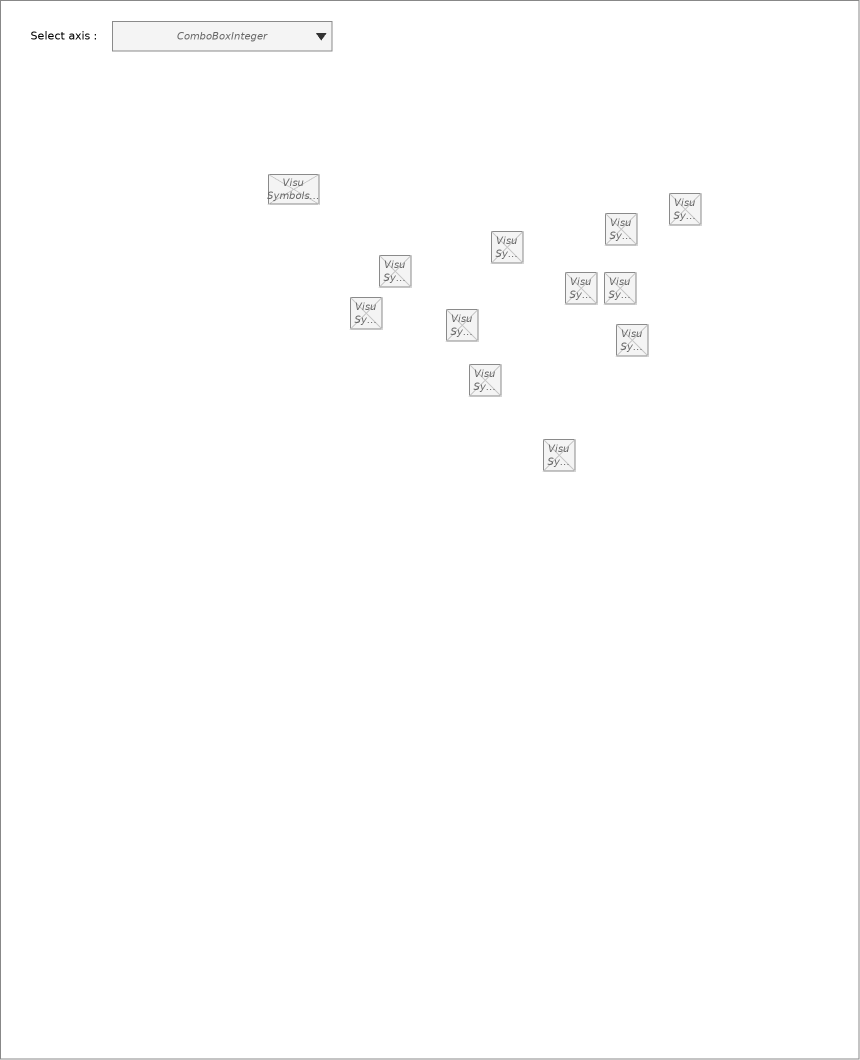
VISUALIZATION VISU_AxisManual  // 860x1060
    Label (22,21 84x30), "Select axis :"
    ComboBoxInteger (112,21 220x30), variable: HMI.iSelectJogAxis
    Image (268,174 51x30), image: VisuSymbols.Symbols.ForwardStandard
    Image (350,297 32x32), image: VisuSymbols.Symbols.Home
    Image (469,364 32x32), image: VisuSymbols.Symbols.Humidity
    Image (543,439 32x32), image: VisuSymbols.Symbols.Keeper
    Image (446,309 32x32), image: VisuSymbols.Symbols.ListNumbers
    Image (604,272 32x32), image: VisuSymbols.Symbols.Marker+
    Image (565,272 32x32), image: VisuSymbols.Symbols.Marker-
    Image (616,324 32x32), image: VisuSymbols.Symbols.Micro
    Image (605,213 32x32), image: VisuSymbols.Symbols.MonitorCurve
    Image (491,231 32x32), image: VisuSymbols.Symbols.Play
    Image (669,193 32x32), image: VisuSymbols.Symbols.Security
    Image (379,255 32x32), image: VisuSymbols.Symbols.Stop
END_VISUALIZATION

(* stored: Version 1.1.0.1, ProductVersion 3.1.4024.6
   Visu VISU_AxisManual: Id {3b5d7614-e3c1-468d-a730-07dedf3e7d48} *)
